// TIA Portal V17 export
// export: Created 2025-06-26T06:49:27.9556467Z, ExportSetting WithDefaults, DisplayName Totally Integrated Automation Portal, DisplayVersion V17 Update 8, DisplayName TIA Portal Openness, DisplayVersion V17 Update 8, DisplayName TIA Portal Version Control Interface, DisplayVersion V17, DisplayName STEP 7 Professional, DisplayVersion V17 Update 8, DisplayName STEP 7 Safety, DisplayVersion V17 Update 6, DisplayName WinCC Advanced, DisplayVersion V17 Update 8
TYPE "stDigitalAlarm"
// stored: IsFailsafeCompliant false
   STRUCT
      bEnable : Bool := true;   // 1 = enabled, 0 = blocked
      bInput : Bool;   // 1 = active, 0 = not active
      tActivationDelay : Time;   // Alarm activation delay
      sState : "stAlarmState";   // Alarm
   END_STRUCT;
END_TYPE
